DATA_BLOCK "dbArchiveControlBoiler"
{ S7_Optimized_Access := 'TRUE' }
VERSION : 0.8
"fbArchiveControlBoiler"

BEGIN

END_DATA_BLOCK

